KUKA KRL data list: geometrylib.dat

&ACCESS RV
&PARAM EDITMASK = *
&PARAM TEMPLATE = C:\KRC\Roboter\Template\vorgabe
DEFDAT geometrylib PUBLIC
   ; Author:      Davide Rosa
   ; e-mail:      dddomodossola@gmail.com
   ; repository:  https://github.com/skilledAutomation/kuka_krl_wonderlibrary

   ; DESCRIPTION:
   ; This library provides geometric data structures and funcions
   ;   For 2D and 3D primitives, the plane is X/Y

   REAL M_PI = 3.1415926535

   global STRUC STR_LINE2D REAL A, B, C, M, Q

   global STRUC STR_CIRCUMFERENCE2D REAL A, B, C

   global STRUC STR_PLANE REAL A, B, C, D ;ax + by + cz + d = 0

   ;In the orthonormal reference system RC(O,i,j,k)
   ;  a vector is identified as:
   ;      v = l*i + m*j + n*k
   global STRUC STR_VECTOR3D REAL L, M, N

   global STRUC STR_LINE3D STR_PLANE plane1, plane2, E6POS point, STR_VECTOR3D vec

ENDDAT
